// TIA Portal V20 export
TYPE "typeCmInterfaceBrakeTest"
// stored: Access Published, Namespace Unit1.Em6
   STRUCT
      visionUnit : "LER_typeBrakeTestEmInterface";
   END_STRUCT;
END_TYPE
